  [1266] = {j1=-10.864, j2=61.673, j3=49.557, j4=-4.156, j5=76.153, j6=-10.598}
  [1267] = {j1=-10.843, j2=62.170, j3=49.109, j4=-4.208, j5=76.502, j6=-10.179}
  [1268] = {j1=-10.824, j2=62.663, j3=48.670, j4=-4.258, j5=76.846, j6=-9.764}
  [1269] = {j1=-10.807, j2=63.152, j3=48.234, j4=-4.302, j5=77.191, j6=-9.351}
  [1270] = {j1=-10.792, j2=63.641, j3=47.799, j4=-4.338, j5=77.541, j6=-8.940}
  [1271] = {j1=-10.790, j2=63.726, j3=47.722, j4=-4.344, j5=77.602, j6=-8.868}
  [1272] = {j1=-10.774, j2=64.208, j3=47.297, j4=-4.390, j5=77.944, j6=-8.456}
  [1273] = {j1=-10.750, j2=64.740, j3=46.858, j4=-4.470, j5=78.272, j6=-8.000}
  [1274] = {j1=-10.722, j2=65.202, j3=46.548, j4=-4.577, j5=78.439, j6=-7.623}
  [1275] = {j1=-10.698, j2=65.509, j3=46.425, j4=-4.679, j5=78.409, j6=-7.406}
  [1276] = {j1=-10.673, j2=65.756, j3=46.411, j4=-4.789, j5=78.237, j6=-7.269}
  [1277] = {j1=-10.648, j2=65.950, j3=46.489, j4=-4.909, j5=77.942, j6=-7.202}
  [1278] = {j1=-10.622, j2=66.101, j3=46.643, j4=-5.043, j5=77.544, j6=-7.192}
  [1279] = {j1=-10.592, j2=66.217, j3=46.855, j4=-5.194, j5=77.062, j6=-7.226}
  [1280] = {j1=-10.560, j2=66.305, j3=47.110, j4=-5.365, j5=76.516, j6=-7.293}
  [1281] = {j1=-10.559, j2=66.323, j3=47.079, j4=-5.369, j5=76.573, j6=-7.250}
  [1282] = {j1=-10.592, j2=66.234, j3=46.825, j4=-5.197, j5=77.118, j6=-7.185}
  [1283] = {j1=-10.621, j2=66.118, j3=46.614, j4=-5.046, j5=77.597, j6=-7.152}
  [1284] = {j1=-10.648, j2=65.966, j3=46.461, j4=-4.911, j5=77.993, j6=-7.164}
  [1285] = {j1=-10.673, j2=65.772, j3=46.384, j4=-4.789, j5=78.286, j6=-7.233}
  [1286] = {j1=-10.698, j2=65.525, j3=46.397, j4=-4.678, j5=78.458, j6=-7.370}
  [1287] = {j1=-10.723, j2=65.219, j3=46.519, j4=-4.575, j5=78.489, j6=-7.588}
  [1288] = {j1=-10.751, j2=64.758, j3=46.827, j4=-4.466, j5=78.325, j6=-7.964}
  [1289] = {j1=-10.775, j2=64.227, j3=47.262, j4=-4.386, j5=78.001, j6=-8.418}
  [1290] = {j1=-10.791, j2=63.747, j3=47.686, j4=-4.339, j5=77.662, j6=-8.829}
  [1291] = {j1=-10.794, j2=63.662, j3=47.761, j4=-4.333, j5=77.600, j6=-8.900}
  [1292] = {j1=-10.808, j2=63.174, j3=48.196, j4=-4.297, j5=77.252, j6=-9.311}
  [1293] = {j1=-10.825, j2=62.685, j3=48.631, j4=-4.253, j5=76.907, j6=-9.723}
  [1294] = {j1=-10.844, j2=62.192, j3=49.070, j4=-4.203, j5=76.562, j6=-10.139}
  [1295] = {j1=-10.865, j2=61.695, j3=49.519, j4=-4.150, j5=76.213, j6=-10.558}
  [1296] = {j1=-10.888, j2=61.189, j3=49.980, j4=-4.096, j5=75.855, j6=-10.983}
  [1297] = {j1=-10.912, j2=60.674, j3=50.459, j4=-4.041, j5=75.484, j6=-11.413}
  [1298] = {j1=-10.936, j2=60.147, j3=50.960, j4=-3.988, j5=75.096, j6=-11.850}
  [1299] = {j1=-10.956, j2=59.676, j3=51.416, j4=-3.950, j5=74.742, j6=-12.232}
  [1300] = {j1=-10.973, j2=59.205, j3=51.873, j4=-3.926, j5=74.393, j6=-12.600}
  [1301] = {j1=-10.987, j2=58.744, j3=52.313, j4=-3.913, j5=74.070, j6=-12.944}
  [1302] = {j1=-10.997, j2=58.303, j3=52.716, j4=-3.909, j5=73.795, j6=-13.252}
  [1303] = {j1=-10.998, j2=58.287, j3=52.730, j4=-3.909, j5=73.786, j6=-13.262}
  [1304] = {j1=-10.999, j2=58.315, j3=52.679, j4=-3.904, j5=73.859, j6=-13.219}
  [1305] = {j1=-10.998, j2=58.331, j3=52.666, j4=-3.904, j5=73.868, j6=-13.209}
  [1306] = {j1=-10.988, j2=58.771, j3=52.265, j4=-3.907, j5=74.140, j6=-12.902}
  [1307] = {j1=-10.974, j2=59.231, j3=51.828, j4=-3.920, j5=74.460, j6=-12.560}
  [1308] = {j1=-10.957, j2=59.701, j3=51.373, j4=-3.944, j5=74.807, j6=-12.193}
  [1309] = {j1=-10.937, j2=60.171, j3=50.919, j4=-3.982, j5=75.158, j6=-11.812}
  [1310] = {j1=-10.913, j2=60.697, j3=50.419, j4=-4.035, j5=75.545, j6=-11.375}
  [1311] = {j1=-10.889, j2=61.212, j3=49.940, j4=-4.090, j5=75.916, j6=-10.944}
  [1312] = {j1=-10.866, j2=61.717, j3=49.479, j4=-4.146, j5=76.274, j6=-10.519}
  [1313] = {j1=-10.845, j2=62.215, j3=49.031, j4=-4.199, j5=76.624, j6=-10.099}
  [1314] = {j1=-10.826, j2=62.707, j3=48.591, j4=-4.248, j5=76.969, j6=-9.683}
  [1315] = {j1=-10.809, j2=63.196, j3=48.158, j4=-4.292, j5=77.312, j6=-9.270}
  [1316] = {j1=-10.795, j2=63.683, j3=47.725, j4=-4.328, j5=77.659, j6=-8.861}
  [1317] = {j1=-10.793, j2=63.768, j3=47.650, j4=-4.334, j5=77.720, j6=-8.789}
  [1318] = {j1=-10.776, j2=64.246, j3=47.230, j4=-4.380, j5=78.055, j6=-8.381}
  [1319] = {j1=-10.752, j2=64.774, j3=46.798, j4=-4.462, j5=78.375, j6=-7.928}
  [1320] = {j1=-10.723, j2=65.233, j3=46.494, j4=-4.572, j5=78.535, j6=-7.553}
  [1321] = {j1=-10.699, j2=65.539, j3=46.373, j4=-4.676, j5=78.503, j6=-7.335}
  [1322] = {j1=-10.674, j2=65.785, j3=46.360, j4=-4.789, j5=78.331, j6=-7.196}
  [1323] = {j1=-10.648, j2=65.980, j3=46.438, j4=-4.912, j5=78.038, j6=-7.126}
  [1324] = {j1=-10.621, j2=66.132, j3=46.590, j4=-5.048, j5=77.643, j6=-7.113}
  [1325] = {j1=-10.591, j2=66.248, j3=46.801, j4=-5.200, j5=77.165, j6=-7.144}
  [1326] = {j1=-10.558, j2=66.337, j3=47.054, j4=-5.373, j5=76.622, j6=-7.207}
  [1327] = {j1=-10.557, j2=66.364, j3=47.008, j4=-5.379, j5=76.709, j6=-7.143}
  [1328] = {j1=-10.590, j2=66.274, j3=46.756, j4=-5.205, j5=77.248, j6=-7.082}
  [1329] = {j1=-10.620, j2=66.157, j3=46.547, j4=-5.052, j5=77.723, j6=-7.054}
  [1330] = {j1=-10.648, j2=66.004, j3=46.396, j4=-4.914, j5=78.115, j6=-7.070}
  [1331] = {j1=-10.674, j2=65.809, j3=46.319, j4=-4.789, j5=78.406, j6=-7.142}
  [1332] = {j1=-10.699, j2=65.563, j3=46.332, j4=-4.675, j5=78.577, j6=-7.282}
  [1333] = {j1=-10.724, j2=65.258, j3=46.451, j4=-4.569, j5=78.611, j6=-7.501}
  [1334] = {j1=-10.754, j2=64.801, j3=46.751, j4=-4.456, j5=78.455, j6=-7.875}
  [1335] = {j1=-10.778, j2=64.276, j3=47.178, j4=-4.373, j5=78.141, j6=-8.324}
  [1336] = {j1=-10.794, j2=63.799, j3=47.594, j4=-4.327, j5=77.809, j6=-8.731}
  [1337] = {j1=-10.797, j2=63.715, j3=47.669, j4=-4.321, j5=77.749, j6=-8.802}
  [1338] = {j1=-10.811, j2=63.229, j3=48.099, j4=-4.285, j5=77.404, j6=-9.210}
  [1339] = {j1=-10.828, j2=62.740, j3=48.533, j4=-4.241, j5=77.060, j6=-9.623}
  [1340] = {j1=-10.847, j2=62.248, j3=48.972, j4=-4.191, j5=76.714, j6=-10.039}
  [1341] = {j1=-10.868, j2=61.749, j3=49.422, j4=-4.138, j5=76.363, j6=-10.461}
  [1342] = {j1=-10.891, j2=61.244, j3=49.884, j4=-4.083, j5=76.003, j6=-10.887}
  [1343] = {j1=-10.915, j2=60.729, j3=50.363, j4=-4.027, j5=75.632, j6=-11.318}
  [1344] = {j1=-10.940, j2=60.203, j3=50.861, j4=-3.973, j5=75.246, j6=-11.755}
  [1345] = {j1=-10.960, j2=59.734, j3=51.313, j4=-3.935, j5=74.897, j6=-12.135}
  [1346] = {j1=-10.976, j2=59.266, j3=51.765, j4=-3.910, j5=74.554, j6=-12.500}
  [1347] = {j1=-10.990, j2=58.808, j3=52.199, j4=-3.898, j5=74.237, j6=-12.840}
  [1348] = {j1=-11.000, j2=58.369, j3=52.597, j4=-3.895, j5=73.967, j6=-13.144}
  [1349] = {j1=-11.000, j2=58.354, j3=52.611, j4=-3.895, j5=73.959, j6=-13.154}
  [1350] = {j1=-11.002, j2=58.398, j3=52.533, j4=-3.888, j5=74.070, j6=-13.089}
  [1351] = {j1=-11.001, j2=58.413, j3=52.520, j4=-3.888, j5=74.078, j6=-13.078}
  [1352] = {j1=-10.991, j2=58.849, j3=52.125, j4=-3.890, j5=74.344, j6=-12.777}
  [1353] = {j1=-10.978, j2=59.305, j3=51.696, j4=-3.902, j5=74.655, j6=-12.440}
  [1354] = {j1=-10.962, j2=59.771, j3=51.248, j4=-3.926, j5=74.993, j6=-12.077}
  [1355] = {j1=-10.942, j2=60.238, j3=50.800, j4=-3.964, j5=75.338, j6=-11.698}
  [1356] = {j1=-10.917, j2=60.762, j3=50.303, j4=-4.019, j5=75.722, j6=-11.262}
  [1357] = {j1=-10.893, j2=61.277, j3=49.825, j4=-4.075, j5=76.093, j6=-10.830}
  [1358] = {j1=-10.870, j2=61.783, j3=49.363, j4=-4.131, j5=76.454, j6=-10.403}
  [1359] = {j1=-10.848, j2=62.281, j3=48.913, j4=-4.184, j5=76.806, j6=-9.980}
  [1360] = {j1=-10.829, j2=62.774, j3=48.474, j4=-4.234, j5=77.152, j6=-9.562}
  [1361] = {j1=-10.812, j2=63.261, j3=48.042, j4=-4.278, j5=77.495, j6=-9.150}
  [1362] = {j1=-10.798, j2=63.746, j3=47.614, j4=-4.313, j5=77.837, j6=-8.743}
  [1363] = {j1=-10.796, j2=63.830, j3=47.539, j4=-4.319, j5=77.897, j6=-8.672}
  [1364] = {j1=-10.780, j2=64.304, j3=47.127, j4=-4.366, j5=78.224, j6=-8.268}
  [1365] = {j1=-10.755, j2=64.826, j3=46.707, j4=-4.450, j5=78.531, j6=-7.821}
  [1366] = {j1=-10.726, j2=65.281, j3=46.411, j4=-4.565, j5=78.682, j6=-7.448}
  [1367] = {j1=-10.700, j2=65.584, j3=46.295, j4=-4.673, j5=78.646, j6=-7.229}
  [1368] = {j1=-10.674, j2=65.830, j3=46.283, j4=-4.789, j5=78.474, j6=-7.088}
  [1369] = {j1=-10.648, j2=66.025, j3=46.360, j4=-4.916, j5=78.184, j6=-7.014}
  [1370] = {j1=-10.620, j2=66.178, j3=46.510, j4=-5.054, j5=77.794, j6=-6.995}
  [1371] = {j1=-10.589, j2=66.296, j3=46.718, j4=-5.210, j5=77.322, j6=-7.020}
  [1372] = {j1=-10.556, j2=66.386, j3=46.969, j4=-5.385, j5=76.785, j6=-7.078}
  [1373] = {j1=-10.555, j2=66.413, j3=46.922, j4=-5.391, j5=76.872, j6=-7.014}
  [1374] = {j1=-10.588, j2=66.322, j3=46.672, j4=-5.215, j5=77.405, j6=-6.959}
  [1375] = {j1=-10.619, j2=66.203, j3=46.466, j4=-5.058, j5=77.874, j6=-6.936}
  [1376] = {j1=-10.647, j2=66.049, j3=46.318, j4=-4.918, j5=78.261, j6=-6.957}
  [1377] = {j1=-10.674, j2=65.854, j3=46.242, j4=-4.790, j5=78.549, j6=-7.033}
  [1378] = {j1=-10.700, j2=65.608, j3=46.253, j4=-4.672, j5=78.721, j6=-7.176}
  [1379] = {j1=-10.727, j2=65.305, j3=46.368, j4=-4.561, j5=78.758, j6=-7.395}
  [1380] = {j1=-10.757, j2=64.854, j3=46.659, j4=-4.444, j5=78.612, j6=-7.766}
  [1381] = {j1=-10.782, j2=64.334, j3=47.075, j4=-4.359, j5=78.310, j6=-8.211}
  [1382] = {j1=-10.798, j2=63.862, j3=47.483, j4=-4.312, j5=77.986, j6=-8.613}
  [1383] = {j1=-10.800, j2=63.778, j3=47.557, j4=-4.306, j5=77.927, j6=-8.683}
  [1384] = {j1=-10.814, j2=63.294, j3=47.984, j4=-4.271, j5=77.586, j6=-9.090}
  [1385] = {j1=-10.831, j2=62.806, j3=48.416, j4=-4.227, j5=77.243, j6=-9.502}
  [1386] = {j1=-10.850, j2=62.313, j3=48.856, j4=-4.177, j5=76.895, j6=-9.921}
  [1387] = {j1=-10.871, j2=61.814, j3=49.307, j4=-4.123, j5=76.540, j6=-10.345}
  [1388] = {j1=-10.894, j2=61.308, j3=49.770, j4=-4.067, j5=76.178, j6=-10.773}
  [1389] = {j1=-10.919, j2=60.793, j3=50.249, j4=-4.010, j5=75.807, j6=-11.206}
  [1390] = {j1=-10.944, j2=60.269, j3=50.744, j4=-3.955, j5=75.424, j6=-11.642}
  [1391] = {j1=-10.964, j2=59.804, j3=51.189, j4=-3.916, j5=75.082, j6=-12.019}
  [1392] = {j1=-10.981, j2=59.340, j3=51.633, j4=-3.892, j5=74.748, j6=-12.379}
  [1393] = {j1=-10.993, j2=58.886, j3=52.059, j4=-3.880, j5=74.441, j6=-12.713}
  [1394] = {j1=-11.003, j2=58.452, j3=52.449, j4=-3.880, j5=74.180, j6=-13.011}
  [1395] = {j1=-11.003, j2=58.437, j3=52.463, j4=-3.880, j5=74.171, j6=-13.022}
  [1396] = {j1=-11.004, j2=58.482, j3=52.382, j4=-3.872, j5=74.286, j6=-12.953}
  [1397] = {j1=-11.004, j2=58.497, j3=52.369, j4=-3.872, j5=74.294, j6=-12.943}
  [1398] = {j1=-10.995, j2=58.929, j3=51.983, j4=-3.872, j5=74.550, j6=-12.648}
  [1399] = {j1=-10.982, j2=59.380, j3=51.563, j4=-3.883, j5=74.851, j6=-12.317}
  [1400] = {j1=-10.966, j2=59.841, j3=51.124, j4=-3.907, j5=75.179, j6=-11.961}
  [1401] = {j1=-10.946, j2=60.303, j3=50.683, j4=-3.947, j5=75.516, j6=-11.585}
  [1402] = {j1=-10.921, j2=60.826, j3=50.190, j4=-4.002, j5=75.896, j6=-11.150}
  [1403] = {j1=-10.896, j2=61.340, j3=49.713, j4=-4.059, j5=76.267, j6=-10.717}
  [1404] = {j1=-10.873, j2=61.847, j3=49.250, j4=-4.116, j5=76.629, j6=-10.287}
  [1405] = {j1=-10.852, j2=62.346, j3=48.798, j4=-4.170, j5=76.985, j6=-9.862}
  [1406] = {j1=-10.833, j2=62.839, j3=48.358, j4=-4.220, j5=77.334, j6=-9.442}
  [1407] = {j1=-10.816, j2=63.327, j3=47.926, j4=-4.263, j5=77.677, j6=-9.029}
  [1408] = {j1=-10.802, j2=63.809, j3=47.502, j4=-4.299, j5=78.015, j6=-8.624}
  [1409] = {j1=-10.800, j2=63.893, j3=47.429, j4=-4.305, j5=78.074, j6=-8.554}
  [1410] = {j1=-10.784, j2=64.362, j3=47.025, j4=-4.352, j5=78.392, j6=-8.154}
  [1411] = {j1=-10.759, j2=64.879, j3=46.615, j4=-4.438, j5=78.687, j6=-7.712}
  [1412] = {j1=-10.728, j2=65.328, j3=46.329, j4=-4.557, j5=78.828, j6=-7.342}
  [1413] = {j1=-10.701, j2=65.629, j3=46.216, j4=-4.670, j5=78.789, j6=-7.122}
  [1414] = {j1=-10.674, j2=65.874, j3=46.206, j4=-4.790, j5=78.617, j6=-6.978}
  [1415] = {j1=-10.647, j2=66.070, j3=46.282, j4=-4.919, j5=78.330, j6=-6.900}
  [1416] = {j1=-10.619, j2=66.224, j3=46.430, j4=-5.061, j5=77.944, j6=-6.876}
  [1417] = {j1=-10.588, j2=66.344, j3=46.635, j4=-5.219, j5=77.478, j6=-6.896}
  [1418] = {j1=-10.554, j2=66.436, j3=46.883, j4=-5.396, j5=76.948, j6=-6.949}
  [1419] = {j1=-10.552, j2=66.463, j3=46.836, j4=-5.403, j5=77.036, j6=-6.883}
  [1420] = {j1=-10.587, j2=66.370, j3=46.589, j4=-5.224, j5=77.563, j6=-6.834}
  [1421] = {j1=-10.618, j2=66.250, j3=46.386, j4=-5.065, j5=78.025, j6=-6.817}
  [1422] = {j1=-10.647, j2=66.095, j3=46.240, j4=-4.921, j5=78.407, j6=-6.843}
  [1423] = {j1=-10.675, j2=65.898, j3=46.164, j4=-4.790, j5=78.692, j6=-6.924}
  [1424] = {j1=-10.702, j2=65.653, j3=46.174, j4=-4.668, j5=78.863, j6=-7.069}
  [1425] = {j1=-10.729, j2=65.353, j3=46.285, j4=-4.554, j5=78.904, j6=-7.289}
  [1426] = {j1=-10.760, j2=64.906, j3=46.568, j4=-4.433, j5=78.768, j6=-7.657}
  [1427] = {j1=-10.785, j2=64.392, j3=46.973, j4=-4.345, j5=78.478, j6=-8.096}
  [1428] = {j1=-10.802, j2=63.925, j3=47.373, j4=-4.297, j5=78.163, j6=-8.494}
  [1429] = {j1=-10.804, j2=63.841, j3=47.446, j4=-4.292, j5=78.105, j6=-8.564}
  [1430] = {j1=-10.818, j2=63.359, j3=47.869, j4=-4.256, j5=77.767, j6=-8.969}
  [1431] = {j1=-10.834, j2=62.872, j3=48.301, j4=-4.213, j5=77.423, j6=-9.382}
  [1432] = {j1=-10.854, j2=62.378, j3=48.743, j4=-4.163, j5=77.072, j6=-9.803}
  [1433] = {j1=-10.875, j2=61.877, j3=49.196, j4=-4.108, j5=76.714, j6=-10.230}
  [1434] = {j1=-10.898, j2=61.370, j3=49.660, j4=-4.051, j5=76.349, j6=-10.661}
  [1435] = {j1=-10.923, j2=60.856, j3=50.138, j4=-3.994, j5=75.978, j6=-11.095}
  [1436] = {j1=-10.948, j2=60.334, j3=50.628, j4=-3.937, j5=75.600, j6=-11.529}
  [1437] = {j1=-10.968, j2=59.873, j3=51.066, j4=-3.898, j5=75.266, j6=-11.902}
  [1438] = {j1=-10.985, j2=59.415, j3=51.500, j4=-3.874, j5=74.944, j6=-12.255}
  [1439] = {j1=-10.997, j2=58.967, j3=51.915, j4=-3.863, j5=74.649, j6=-12.582}
  [1440] = {j1=-11.006, j2=58.537, j3=52.297, j4=-3.864, j5=74.397, j6=-12.874}
  [1441] = {j1=-11.006, j2=58.522, j3=52.311, j4=-3.864, j5=74.388, j6=-12.884}
  [1442] = {j1=-11.007, j2=58.569, j3=52.226, j4=-3.857, j5=74.507, j6=-12.814}
  [1443] = {j1=-11.007, j2=58.584, j3=52.214, j4=-3.857, j5=74.514, j6=-12.804}
  [1444] = {j1=-10.998, j2=59.011, j3=51.837, j4=-3.855, j5=74.760, j6=-12.516}
  [1445] = {j1=-10.986, j2=59.455, j3=51.428, j4=-3.865, j5=75.048, j6=-12.193}
  [1446] = {j1=-10.970, j2=59.910, j3=51.001, j4=-3.889, j5=75.363, j6=-11.843}
  [1447] = {j1=-10.950, j2=60.368, j3=50.568, j4=-3.929, j5=75.691, j6=-11.473}
  [1448] = {j1=-10.925, j2=60.888, j3=50.081, j4=-3.986, j5=76.065, j6=-11.040}
  [1449] = {j1=-10.900, j2=61.402, j3=49.605, j4=-4.044, j5=76.435, j6=-10.606}
  [1450] = {j1=-10.877, j2=61.909, j3=49.140, j4=-4.101, j5=76.801, j6=-10.173}
  [1451] = {j1=-10.855, j2=62.410, j3=48.686, j4=-4.155, j5=77.160, j6=-9.745}
  [1452] = {j1=-10.836, j2=62.904, j3=48.244, j4=-4.205, j5=77.512, j6=-9.322}
  [1453] = {j1=-10.819, j2=63.392, j3=47.812, j4=-4.249, j5=77.857, j6=-8.908}
  [1454] = {j1=-10.806, j2=63.872, j3=47.391, j4=-4.284, j5=78.192, j6=-8.504}
  [1455] = {j1=-10.803, j2=63.955, j3=47.320, j4=-4.290, j5=78.249, j6=-8.434}
  [1456] = {j1=-10.787, j2=64.420, j3=46.923, j4=-4.338, j5=78.559, j6=-8.039}
  [1457] = {j1=-10.762, j2=64.931, j3=46.524, j4=-4.427, j5=78.843, j6=-7.602}
  [1458] = {j1=-10.730, j2=65.375, j3=46.247, j4=-4.550, j5=78.974, j6=-7.235}
  [1459] = {j1=-10.702, j2=65.674, j3=46.138, j4=-4.666, j5=78.930, j6=-7.015}
  [1460] = {j1=-10.675, j2=65.918, j3=46.129, j4=-4.790, j5=78.759, j6=-6.868}
  [1461] = {j1=-10.647, j2=66.115, j3=46.205, j4=-4.922, j5=78.475, j6=-6.786}
  [1462] = {j1=-10.618, j2=66.270, j3=46.350, j4=-5.067, j5=78.095, j6=-6.757}
  [1463] = {j1=-10.586, j2=66.392, j3=46.552, j4=-5.227, j5=77.635, j6=-6.771}
  [1464] = {j1=-10.552, j2=66.485, j3=46.798, j4=-5.407, j5=77.110, j6=-6.818}
  [1465] = {j1=-10.550, j2=66.513, j3=46.749, j4=-5.413, j5=77.199, j6=-6.752}
  [1466] = {j1=-10.585, j2=66.419, j3=46.506, j4=-5.232, j5=77.720, j6=-6.708}
  [1467] = {j1=-10.617, j2=66.296, j3=46.306, j4=-5.071, j5=78.176, j6=-6.697}
  [1468] = {j1=-10.647, j2=66.140, j3=46.162, j4=-4.924, j5=78.553, j6=-6.728}
  [1469] = {j1=-10.675, j2=65.943, j3=46.087, j4=-4.790, j5=78.834, j6=-6.813}
  [1470] = {j1=-10.703, j2=65.698, j3=46.096, j4=-4.665, j5=79.005, j6=-6.961}
  [1471] = {j1=-10.731, j2=65.400, j3=46.203, j4=-4.546, j5=79.050, j6=-7.181}
  [1472] = {j1=-10.763, j2=64.958, j3=46.476, j4=-4.421, j5=78.923, j6=-7.547}
  [1473] = {j1=-10.789, j2=64.450, j3=46.871, j4=-4.331, j5=78.645, j6=-7.981}
  [1474] = {j1=-10.805, j2=63.987, j3=47.264, j4=-4.283, j5=78.338, j6=-8.374}
  [1475] = {j1=-10.807, j2=63.904, j3=47.336, j4=-4.277, j5=78.281, j6=-8.444}
  [1476] = {j1=-10.821, j2=63.423, j3=47.756, j4=-4.242, j5=77.946, j6=-8.847}
  [1477] = {j1=-10.838, j2=62.935, j3=48.188, j4=-4.198, j5=77.600, j6=-9.263}
  [1478] = {j1=-10.857, j2=62.440, j3=48.632, j4=-4.148, j5=77.245, j6=-9.687}
  [1479] = {j1=-10.879, j2=61.938, j3=49.088, j4=-4.093, j5=76.882, j6=-10.117}
  [1480] = {j1=-10.902, j2=61.430, j3=49.554, j4=-4.035, j5=76.515, j6=-10.551}
  [1481] = {j1=-10.927, j2=60.916, j3=50.030, j4=-3.977, j5=76.144, j6=-10.985}
  [1482] = {j1=-10.952, j2=60.398, j3=50.515, j4=-3.920, j5=75.772, j6=-11.417}
  [1483] = {j1=-10.972, j2=59.942, j3=50.944, j4=-3.880, j5=75.450, j6=-11.784}
  [1484] = {j1=-10.988, j2=59.490, j3=51.366, j4=-3.856, j5=75.141, j6=-12.130}
  [1485] = {j1=-11.000, j2=59.049, j3=51.769, j4=-3.846, j5=74.859, j6=-12.448}
  [1486] = {j1=-11.008, j2=58.625, j3=52.141, j4=-3.848, j5=74.619, j6=-12.733}
  [1487] = {j1=-11.009, j2=58.610, j3=52.154, j4=-3.848, j5=74.610, j6=-12.743}
  [1488] = {j1=-11.010, j2=58.659, j3=52.067, j4=-3.841, j5=74.732, j6=-12.670}
  [1489] = {j1=-11.009, j2=58.674, j3=52.054, j4=-3.841, j5=74.739, j6=-12.660}
  [1490] = {j1=-11.002, j2=59.094, j3=51.689, j4=-3.838, j5=74.973, j6=-12.380}
  [1491] = {j1=-10.990, j2=59.531, j3=51.293, j4=-3.847, j5=75.246, j6=-12.066}
  [1492] = {j1=-10.974, j2=59.979, j3=50.878, j4=-3.871, j5=75.546, j6=-11.724}
  [1493] = {j1=-10.954, j2=60.432, j3=50.455, j4=-3.911, j5=75.862, j6=-11.360}
  [1494] = {j1=-10.929, j2=60.948, j3=49.974, j4=-3.969, j5=76.230, j6=-10.930}
  [1495] = {j1=-10.904, j2=61.461, j3=49.500, j4=-4.027, j5=76.599, j6=-10.496}
  [1496] = {j1=-10.881, j2=61.969, j3=49.033, j4=-4.085, j5=76.968, j6=-10.061}
  [1497] = {j1=-10.859, j2=62.472, j3=48.577, j4=-4.140, j5=77.331, j6=-9.629}
  [1498] = {j1=-10.839, j2=62.967, j3=48.132, j4=-4.191, j5=77.688, j6=-9.203}
  [1499] = {j1=-10.823, j2=63.455, j3=47.700, j4=-4.234, j5=78.034, j6=-8.787}
  [1500] = {j1=-10.809, j2=63.935, j3=47.282, j4=-4.270, j5=78.367, j6=-8.383}
  [1501] = {j1=-10.807, j2=64.017, j3=47.211, j4=-4.275, j5=78.424, j6=-8.314}
  [1502] = {j1=-10.791, j2=64.478, j3=46.822, j4=-4.324, j5=78.725, j6=-7.923}
  [1503] = {j1=-10.765, j2=64.982, j3=46.434, j4=-4.415, j5=78.997, j6=-7.491}
  [1504] = {j1=-10.732, j2=65.422, j3=46.166, j4=-4.542, j5=79.118, j6=-7.127}
  [1505] = {j1=-10.704, j2=65.719, j3=46.061, j4=-4.663, j5=79.072, j6=-6.906}
  [1506] = {j1=-10.675, j2=65.962, j3=46.053, j4=-4.789, j5=78.900, j6=-6.757}
  [1507] = {j1=-10.647, j2=66.159, j3=46.127, j4=-4.925, j5=78.619, j6=-6.671}
  [1508] = {j1=-10.617, j2=66.316, j3=46.271, j4=-5.073, j5=78.244, j6=-6.637}
  [1509] = {j1=-10.585, j2=66.440, j3=46.470, j4=-5.236, j5=77.791, j6=-6.645}
  [1510] = {j1=-10.550, j2=66.535, j3=46.712, j4=-5.418, j5=77.273, j6=-6.686}
  [1511] = {j1=-10.548, j2=66.563, j3=46.663, j4=-5.424, j5=77.363, j6=-6.620}
  [1512] = {j1=-10.584, j2=66.467, j3=46.422, j4=-5.241, j5=77.877, j6=-6.582}
  [1513] = {j1=-10.616, j2=66.342, j3=46.225, j4=-5.076, j5=78.326, j6=-6.576}
  [1514] = {j1=-10.646, j2=66.184, j3=46.084, j4=-4.927, j5=78.698, j6=-6.613}
  [1515] = {j1=-10.675, j2=65.987, j3=46.011, j4=-4.790, j5=78.976, j6=-6.701}
  [1516] = {j1=-10.704, j2=65.743, j3=46.019, j4=-4.661, j5=79.147, j6=-6.852}
  [1517] = {j1=-10.733, j2=65.447, j3=46.122, j4=-4.539, j5=79.194, j6=-7.073}
  [1518] = {j1=-10.766, j2=65.010, j3=46.386, j4=-4.410, j5=79.077, j6=-7.435}
  [1519] = {j1=-10.792, j2=64.508, j3=46.770, j4=-4.317, j5=78.810, j6=-7.864}
  [1520] = {j1=-10.809, j2=64.048, j3=47.156, j4=-4.268, j5=78.511, j6=-8.254}
  [1521] = {j1=-10.811, j2=63.966, j3=47.227, j4=-4.263, j5=78.455, j6=-8.323}
  [1522] = {j1=-10.824, j2=63.487, j3=47.645, j4=-4.227, j5=78.122, j6=-8.727}
  [1523] = {j1=-10.841, j2=62.998, j3=48.078, j4=-4.183, j5=77.773, j6=-9.144}
  [1524] = {j1=-10.861, j2=62.501, j3=48.525, j4=-4.132, j5=77.414, j6=-9.572}
  [1525] = {j1=-10.883, j2=61.997, j3=48.984, j4=-4.077, j5=77.047, j6=-10.005}
  [1526] = {j1=-10.906, j2=61.488, j3=49.452, j4=-4.019, j5=76.676, j6=-10.442}
  [1527] = {j1=-10.931, j2=60.975, j3=49.926, j4=-3.960, j5=76.306, j6=-10.876}
  [1528] = {j1=-10.956, j2=60.460, j3=50.404, j4=-3.902, j5=75.942, j6=-11.304}
  [1529] = {j1=-10.977, j2=60.011, j3=50.822, j4=-3.862, j5=75.632, j6=-11.664}
  [1530] = {j1=-10.992, j2=59.566, j3=51.230, j4=-3.838, j5=75.339, j6=-12.001}
  [1531] = {j1=-11.004, j2=59.133, j3=51.620, j4=-3.829, j5=75.073, j6=-12.310}
  [1532] = {j1=-11.011, j2=58.715, j3=51.980, j4=-3.832, j5=74.845, j6=-12.587}
  [1533] = {j1=-11.011, j2=58.700, j3=51.993, j4=-3.833, j5=74.837, j6=-12.597}
  [1534] = {j1=-11.012, j2=58.746, j3=51.911, j4=-3.827, j5=74.952, j6=-12.528}
  [1535] = {j1=-11.012, j2=58.761, j3=51.899, j4=-3.826, j5=74.958, j6=-12.519}
  [1536] = {j1=-11.005, j2=59.175, j3=51.545, j4=-3.822, j5=75.179, j6=-12.246}
  [1537] = {j1=-10.994, j2=59.604, j3=51.163, j4=-3.831, j5=75.436, j6=-11.942}
  [1538] = {j1=-10.978, j2=60.044, j3=50.762, j4=-3.854, j5=75.720, j6=-11.610}
  [1539] = {j1=-10.958, j2=60.491, j3=50.351, j4=-3.895, j5=76.023, j6=-11.253}
  [1540] = {j1=-10.933, j2=61.003, j3=49.877, j4=-3.953, j5=76.382, j6=-10.827}
  [1541] = {j1=-10.908, j2=61.515, j3=49.404, j4=-4.012, j5=76.751, j6=-10.392}
  [1542] = {j1=-10.884, j2=62.024, j3=48.936, j4=-4.070, j5=77.121, j6=-9.955}
  [1543] = {j1=-10.863, j2=62.528, j3=48.477, j4=-4.126, j5=77.490, j6=-9.520}
  [1544] = {j1=-10.843, j2=63.026, j3=48.029, j4=-4.176, j5=77.851, j6=-9.090}
  [1545] = {j1=-10.826, j2=63.514, j3=47.596, j4=-4.220, j5=78.200, j6=-8.672}
  [1546] = {j1=-10.812, j2=63.993, j3=47.180, j4=-4.256, j5=78.532, j6=-8.268}
  [1547] = {j1=-10.810, j2=64.075, j3=47.110, j4=-4.261, j5=78.587, j6=-8.200}
  [1548] = {j1=-10.794, j2=64.532, j3=46.727, j4=-4.311, j5=78.882, j6=-7.811}
  [1549] = {j1=-10.768, j2=65.031, j3=46.349, j4=-4.404, j5=79.142, j6=-7.384}
  [1550] = {j1=-10.734, j2=65.466, j3=46.089, j4=-4.535, j5=79.255, j6=-7.023}
  [1551] = {j1=-10.705, j2=65.761, j3=45.988, j4=-4.659, j5=79.205, j6=-6.801}
  [1552] = {j1=-10.676, j2=66.004, j3=45.981, j4=-4.789, j5=79.034, j6=-6.650}
  [1553] = {j1=-10.647, j2=66.202, j3=46.054, j4=-4.928, j5=78.756, j6=-6.560}
  [1554] = {j1=-10.616, j2=66.360, j3=46.195, j4=-5.078, j5=78.386, j6=-6.521}
  [1555] = {j1=-10.583, j2=66.485, j3=46.391, j4=-5.243, j5=77.939, j6=-6.524}
  [1556] = {j1=-10.548, j2=66.582, j3=46.631, j4=-5.428, j5=77.427, j6=-6.559}
  [1557] = {j1=-10.547, j2=66.608, j3=46.585, j4=-5.433, j5=77.510, j6=-6.498}
  [1558] = {j1=-10.583, j2=66.510, j3=46.348, j4=-5.247, j5=78.017, j6=-6.465}
  [1559] = {j1=-10.615, j2=66.384, j3=46.154, j4=-5.081, j5=78.461, j6=-6.465}
  [1560] = {j1=-10.646, j2=66.224, j3=46.015, j4=-4.929, j5=78.828, j6=-6.506}
  [1561] = {j1=-10.676, j2=66.026, j3=45.942, j4=-4.789, j5=79.103, j6=-6.599}
  [1562] = {j1=-10.705, j2=65.783, j3=45.950, j4=-4.658, j5=79.273, j6=-6.751}
  [1563] = {j1=-10.735, j2=65.488, j3=46.050, j4=-4.532, j5=79.323, j6=-6.973}
  [1564] = {j1=-10.769, j2=65.055, j3=46.306, j4=-4.399, j5=79.214, j6=-7.333}
  [1565] = {j1=-10.796, j2=64.558, j3=46.681, j4=-4.304, j5=78.958, j6=-7.758}
  [1566] = {j1=-10.812, j2=64.102, j3=47.061, j4=-4.255, j5=78.665, j6=-8.145}
  [1567] = {j1=-10.814, j2=64.020, j3=47.132, j4=-4.249, j5=78.609, j6=-8.214}
  [1568] = {j1=-10.828, j2=63.542, j3=47.547, j4=-4.213, j5=78.277, j6=-8.617}
  [1569] = {j1=-10.845, j2=63.052, j3=47.982, j4=-4.169, j5=77.926, j6=-9.037}
  [1570] = {j1=-10.864, j2=62.554, j3=48.432, j4=-4.118, j5=77.561, j6=-9.468}
  [1571] = {j1=-10.886, j2=62.048, j3=48.894, j4=-4.062, j5=77.190, j6=-9.905}
  [1572] = {j1=-10.910, j2=61.538, j3=49.363, j4=-4.004, j5=76.817, j6=-10.344}
  [1573] = {j1=-10.935, j2=61.026, j3=49.836, j4=-3.944, j5=76.449, j6=-10.778}
  [1574] = {j1=-10.960, j2=60.515, j3=50.307, j4=-3.886, j5=76.092, j6=-11.202}
  [1575] = {j1=-10.980, j2=60.072, j3=50.713, j4=-3.846, j5=75.795, j6=-11.555}
  [1576] = {j1=-10.996, j2=59.635, j3=51.108, j4=-3.822, j5=75.518, j6=-11.882}
  [1577] = {j1=-11.006, j2=59.210, j3=51.483, j4=-3.813, j5=75.269, j6=-12.181}
  [1578] = {j1=-11.013, j2=58.799, j3=51.832, j4=-3.818, j5=75.054, j6=-12.450}
  [1579] = {j1=-11.013, j2=58.784, j3=51.844, j4=-3.818, j5=75.047, j6=-12.459}
  [1580] = {j1=-11.014, j2=58.831, j3=51.759, j4=-3.812, j5=75.164, j6=-12.389}
  [1581] = {j1=-11.014, j2=58.846, j3=51.748, j4=-3.812, j5=75.170, j6=-12.380}
  [1582] = {j1=-11.007, j2=59.253, j3=51.406, j4=-3.807, j5=75.377, j6=-12.116}
  [1583] = {j1=-10.997, j2=59.674, j3=51.039, j4=-3.815, j5=75.616, j6=-11.822}
  [1584] = {j1=-10.982, j2=60.106, j3=50.653, j4=-3.838, j5=75.883, j6=-11.499}
  [1585] = {j1=-10.962, j2=60.545, j3=50.254, j4=-3.879, j5=76.172, j6=-11.150}
  [1586] = {j1=-10.937, j2=61.053, j3=49.788, j4=-3.937, j5=76.523, j6=-10.729}
  [1587] = {j1=-10.912, j2=61.564, j3=49.318, j4=-3.996, j5=76.889, j6=-10.295}
  [1588] = {j1=-10.888, j2=62.074, j3=48.848, j4=-4.055, j5=77.262, j6=-9.856}
  [1589] = {j1=-10.866, j2=62.580, j3=48.386, j4=-4.111, j5=77.635, j6=-9.417}
  [1590] = {j1=-10.846, j2=63.079, j3=47.935, j4=-4.162, j5=78.001, j6=-8.984}
  [1591] = {j1=-10.829, j2=63.569, j3=47.500, j4=-4.206, j5=78.353, j6=-8.563}
  [1592] = {j1=-10.816, j2=64.046, j3=47.085, j4=-4.242, j5=78.685, j6=-8.159}
  [1593] = {j1=-10.814, j2=64.128, j3=47.016, j4=-4.248, j5=78.739, j6=-8.090}
  [1594] = {j1=-10.797, j2=64.582, j3=46.639, j4=-4.298, j5=79.028, j6=-7.705}
  [1595] = {j1=-10.770, j2=65.076, j3=46.270, j4=-4.393, j5=79.279, j6=-7.282}
  [1596] = {j1=-10.736, j2=65.507, j3=46.018, j4=-4.528, j5=79.382, j6=-6.923}
  [1597] = {j1=-10.706, j2=65.800, j3=45.920, j4=-4.655, j5=79.330, j6=-6.701}
  [1598] = {j1=-10.676, j2=66.043, j3=45.914, j4=-4.788, j5=79.159, j6=-6.547}
  [1599] = {j1=-10.646, j2=66.241, j3=45.986, j4=-4.930, j5=78.885, j6=-6.453}
  [1600] = {j1=-10.615, j2=66.401, j3=46.125, j4=-5.082, j5=78.520, j6=-6.409}
  [1601] = {j1=-10.582, j2=66.527, j3=46.318, j4=-5.250, j5=78.078, j6=-6.407}
  [1602] = {j1=-10.546, j2=66.626, j3=46.554, j4=-5.436, j5=77.574, j6=-6.437}
  [1603] = {j1=-10.545, j2=66.652, j3=46.508, j4=-5.441, j5=77.657, j6=-6.375}
  [1604] = {j1=-10.581, j2=66.553, j3=46.274, j4=-5.254, j5=78.158, j6=-6.348}
  [1605] = {j1=-10.615, j2=66.425, j3=46.083, j4=-5.085, j5=78.595, j6=-6.353}
  [1606] = {j1=-10.646, j2=66.264, j3=45.946, j4=-4.931, j5=78.957, j6=-6.399}
  [1607] = {j1=-10.676, j2=66.065, j3=45.875, j4=-4.788, j5=79.229, j6=-6.495}
  [1608] = {j1=-10.707, j2=65.822, j3=45.882, j4=-4.654, j5=79.398, j6=-6.650}
  [1609] = {j1=-10.737, j2=65.529, j3=45.979, j4=-4.525, j5=79.451, j6=-6.872}
  [1610] = {j1=-10.772, j2=65.100, j3=46.228, j4=-4.389, j5=79.350, j6=-7.230}
  [1611] = {j1=-10.799, j2=64.608, j3=46.594, j4=-4.292, j5=79.103, j6=-7.651}
  [1612] = {j1=-10.815, j2=64.155, j3=46.968, j4=-4.241, j5=78.816, j6=-8.036}
  [1613] = {j1=-10.817, j2=64.073, j3=47.038, j4=-4.235, j5=78.761, j6=-8.104}
  [1614] = {j1=-10.831, j2=63.596, j3=47.453, j4=-4.199, j5=78.429, j6=-8.508}
  [1615] = {j1=-10.848, j2=63.105, j3=47.890, j4=-4.155, j5=78.074, j6=-8.931}
  [1616] = {j1=-10.868, j2=62.604, j3=48.344, j4=-4.103, j5=77.704, j6=-9.366}
  [1617] = {j1=-10.890, j2=62.097, j3=48.809, j4=-4.047, j5=77.328, j6=-9.807}
  [1618] = {j1=-10.914, j2=61.586, j3=49.279, j4=-3.988, j5=76.952, j6=-10.247}
  [1619] = {j1=-10.939, j2=61.075, j3=49.749, j4=-3.929, j5=76.586, j6=-10.680}
  [1620] = {j1=-10.964, j2=60.569, j3=50.212, j4=-3.870, j5=76.239, j6=-11.099}
  [1621] = {j1=-10.984, j2=60.133, j3=50.605, j4=-3.830, j5=75.957, j6=-11.444}
  [1622] = {j1=-10.999, j2=59.705, j3=50.984, j4=-3.806, j5=75.698, j6=-11.761}
  [1623] = {j1=-11.009, j2=59.288, j3=51.344, j4=-3.798, j5=75.467, j6=-12.049}
  [1624] = {j1=-11.015, j2=58.884, j3=51.680, j4=-3.804, j5=75.267, j6=-12.309}
  [1625] = {j1=-11.016, j2=58.869, j3=51.692, j4=-3.804, j5=75.259, j6=-12.318}
  [1626] = {j1=-11.016, j2=58.918, j3=51.605, j4=-3.799, j5=75.379, j6=-12.246}
  [1627] = {j1=-11.016, j2=58.932, j3=51.594, j4=-3.798, j5=75.385, j6=-12.237}
  [1628] = {j1=-11.010, j2=59.332, j3=51.265, j4=-3.792, j5=75.577, j6=-11.982}
  [1629] = {j1=-11.000, j2=59.744, j3=50.915, j4=-3.799, j5=75.797, j6=-11.699}
  [1630] = {j1=-10.985, j2=60.166, j3=50.546, j4=-3.823, j5=76.045, j6=-11.388}
  [1631] = {j1=-10.966, j2=60.599, j3=50.160, j4=-3.863, j5=76.318, j6=-11.048}
  [1632] = {j1=-10.941, j2=61.102, j3=49.702, j4=-3.921, j5=76.659, j6=-10.632}
  [1633] = {j1=-10.916, j2=61.611, j3=49.235, j4=-3.981, j5=77.022, j6=-10.199}
  [1634] = {j1=-10.892, j2=62.121, j3=48.765, j4=-4.040, j5=77.398, j6=-9.758}
  [1635] = {j1=-10.870, j2=62.629, j3=48.299, j4=-4.096, j5=77.776, j6=-9.315}
  [1636] = {j1=-10.850, j2=63.131, j3=47.844, j4=-4.147, j5=78.147, j6=-8.878}
  [1637] = {j1=-10.833, j2=63.622, j3=47.407, j4=-4.192, j5=78.503, j6=-8.454}
  [1638] = {j1=-10.819, j2=64.099, j3=46.993, j4=-4.228, j5=78.834, j6=-8.050}
  [1639] = {j1=-10.817, j2=64.180, j3=46.925, j4=-4.234, j5=78.888, j6=-7.982}
  [1640] = {j1=-10.801, j2=64.631, j3=46.554, j4=-4.285, j5=79.171, j6=-7.598}
  [1641] = {j1=-10.773, j2=65.121, j3=46.192, j4=-4.383, j5=79.413, j6=-7.179}
  [1642] = {j1=-10.738, j2=65.547, j3=45.948, j4=-4.521, j5=79.509, j6=-6.822}
  [1643] = {j1=-10.707, j2=65.839, j3=45.853, j4=-4.651, j5=79.454, j6=-6.600}
  [1644] = {j1=-10.677, j2=66.081, j3=45.847, j4=-4.787, j5=79.284, j6=-6.443}
  [1645] = {j1=-10.646, j2=66.280, j3=45.918, j4=-4.931, j5=79.013, j6=-6.345}
  [1646] = {j1=-10.615, j2=66.441, j3=46.054, j4=-5.086, j5=78.653, j6=-6.297}
  [1647] = {j1=-10.581, j2=66.570, j3=46.244, j4=-5.256, j5=78.217, j6=-6.289}
  [1648] = {j1=-10.545, j2=66.670, j3=46.477, j4=-5.444, j5=77.719, j6=-6.313}
  [1649] = {j1=-10.543, j2=66.708, j3=46.412, j4=-5.452, j5=77.837, j6=-6.227}
  [1650] = {j1=-10.580, j2=66.606, j3=46.182, j4=-5.262, j5=78.330, j6=-6.206}
  [1651] = {j1=-10.614, j2=66.476, j3=45.994, j4=-5.090, j5=78.760, j6=-6.218}
  [1652] = {j1=-10.646, j2=66.313, j3=45.861, j4=-4.933, j5=79.115, j6=-6.270}
  [1653] = {j1=-10.677, j2=66.113, j3=45.791, j4=-4.787, j5=79.383, j6=-6.370}
  [1654] = {j1=-10.708, j2=65.871, j3=45.797, j4=-4.649, j5=79.552, j6=-6.528}
  [1655] = {j1=-10.739, j2=65.580, j3=45.891, j4=-4.517, j5=79.607, j6=-6.751}
  [1656] = {j1=-10.775, j2=65.155, j3=46.131, j4=-4.376, j5=79.515, j6=-7.107}
  [1657] = {j1=-10.803, j2=64.669, j3=46.488, j4=-4.277, j5=79.278, j6=-7.524}
  [1658] = {j1=-10.819, j2=64.219, j3=46.856, j4=-4.225, j5=78.998, j6=-7.906}
  [1659] = {j1=-10.821, j2=64.137, j3=46.926, j4=-4.219, j5=78.943, j6=-7.974}
  [1660] = {j1=-10.835, j2=63.660, j3=47.340, j4=-4.183, j5=78.610, j6=-8.379}
  [1661] = {j1=-10.852, j2=63.167, j3=47.780, j4=-4.137, j5=78.250, j6=-8.806}
  [1662] = {j1=-10.873, j2=62.664, j3=48.238, j4=-4.085, j5=77.874, j6=-9.246}
  [1663] = {j1=-10.895, j2=62.154, j3=48.707, j4=-4.029, j5=77.491, j6=-9.691}
  [1664] = {j1=-10.919, j2=61.643, j3=49.179, j4=-3.970, j5=77.113, j6=-10.133}
  [1665] = {j1=-10.943, j2=61.134, j3=49.645, j4=-3.910, j5=76.751, j6=-10.565}
  [1666] = {j1=-10.969, j2=60.634, j3=50.097, j4=-3.852, j5=76.417, j6=-10.977}
  [1667] = {j1=-10.988, j2=60.207, j3=50.473, j4=-3.811, j5=76.154, j6=-11.310}
  [1668] = {j1=-11.002, j2=59.791, j3=50.831, j4=-3.788, j5=75.920, j6=-11.613}
  [1669] = {j1=-11.012, j2=59.385, j3=51.170, j4=-3.781, j5=75.713, j6=-11.887}
  [1670] = {j1=-11.018, j2=58.991, j3=51.489, j4=-3.788, j5=75.531, j6=-12.136}
  [1671] = {j1=-11.018, j2=58.976, j3=51.501, j4=-3.788, j5=75.524, j6=-12.144}
  [1672] = {j1=-11.018, j2=59.011, j3=51.440, j4=-3.784, j5=75.608, j6=-12.094}
  [1673] = {j1=-11.018, j2=59.024, j3=51.430, j4=-3.784, j5=75.613, j6=-12.085}
  [1674] = {j1=-11.013, j2=59.416, j3=51.116, j4=-3.777, j5=75.788, j6=-11.840}
  [1675] = {j1=-11.003, j2=59.817, j3=50.784, j4=-3.784, j5=75.987, j6=-11.570}
  [1676] = {j1=-10.989, j2=60.230, j3=50.433, j4=-3.807, j5=76.213, j6=-11.271}
  [1677] = {j1=-10.970, j2=60.653, j3=50.063, j4=-3.847, j5=76.469, j6=-10.941}
  [1678] = {j1=-10.945, j2=61.151, j3=49.616, j4=-3.905, j5=76.798, j6=-10.532}
  [1679] = {j1=-10.920, j2=61.658, j3=49.152, j4=-3.964, j5=77.158, j6=-10.101}
  [1680] = {j1=-10.896, j2=62.169, j3=48.681, j4=-4.023, j5=77.535, j6=-9.658}
  [1681] = {j1=-10.874, j2=62.679, j3=48.212, j4=-4.080, j5=77.918, j6=-9.211}
  [1682] = {j1=-10.854, j2=63.183, j3=47.753, j4=-4.132, j5=78.295, j6=-8.770}
  [1683] = {j1=-10.837, j2=63.675, j3=47.313, j4=-4.177, j5=78.655, j6=-8.342}
  [1684] = {j1=-10.823, j2=64.152, j3=46.900, j4=-4.214, j5=78.987, j6=-7.937}
  [1685] = {j1=-10.821, j2=64.233, j3=46.831, j4=-4.220, j5=79.041, j6=-7.869}
  [1686] = {j1=-10.804, j2=64.682, j3=46.465, j4=-4.272, j5=79.319, j6=-7.487}
  [1687] = {j1=-10.776, j2=65.166, j3=46.112, j4=-4.372, j5=79.552, j6=-7.071}
  [1688] = {j1=-10.740, j2=65.589, j3=45.875, j4=-4.513, j5=79.641, j6=-6.716}
  [1689] = {j1=-10.709, j2=65.879, j3=45.783, j4=-4.647, j5=79.583, j6=-6.493}
  [1690] = {j1=-10.678, j2=66.121, j3=45.778, j4=-4.786, j5=79.414, j6=-6.334}
  [1691] = {j1=-10.646, j2=66.321, j3=45.847, j4=-4.932, j5=79.147, j6=-6.232}
  [1692] = {j1=-10.614, j2=66.484, j3=45.981, j4=-5.090, j5=78.792, j6=-6.178}
  [1693] = {j1=-10.580, j2=66.614, j3=46.168, j4=-5.262, j5=78.363, j6=-6.165}
  [1694] = {j1=-10.543, j2=66.716, j3=46.397, j4=-5.453, j5=77.871, j6=-6.184}
  [1695] = {j1=-10.542, j2=66.735, j3=46.365, j4=-5.456, j5=77.930, j6=-6.141}
  [1696] = {j1=-10.579, j2=66.632, j3=46.137, j4=-5.265, j5=78.418, j6=-6.124}
  [1697] = {j1=-10.614, j2=66.500, j3=45.952, j4=-5.092, j5=78.844, j6=-6.139}
  [1698] = {j1=-10.646, j2=66.337, j3=45.820, j4=-4.933, j5=79.196, j6=-6.194}
  [1699] = {j1=-10.678, j2=66.136, j3=45.752, j4=-4.785, j5=79.461, j6=-6.297}
  [1700] = {j1=-10.709, j2=65.894, j3=45.758, j4=-4.646, j5=79.629, j6=-6.457}
  [1701] = {j1=-10.741, j2=65.603, j3=45.849, j4=-4.511, j5=79.686, j6=-6.681}
  [1702] = {j1=-10.777, j2=65.182, j3=46.086, j4=-4.368, j5=79.598, j6=-7.035}
  [1703] = {j1=-10.805, j2=64.697, j3=46.437, j4=-4.267, j5=79.366, j6=-7.450}
  [1704] = {j1=-10.822, j2=64.249, j3=46.803, j4=-4.215, j5=79.088, j6=-7.831}
  [1705] = {j1=-10.824, j2=64.168, j3=46.872, j4=-4.208, j5=79.034, j6=-7.900}
  [1706] = {j1=-10.838, j2=63.690, j3=47.287, j4=-4.172, j5=78.700, j6=-8.306}
  [1707] = {j1=-10.855, j2=63.197, j3=47.728, j4=-4.126, j5=78.337, j6=-8.735}
  [1708] = {j1=-10.876, j2=62.692, j3=48.189, j4=-4.074, j5=77.957, j6=-9.177}
  [1709] = {j1=-10.898, j2=62.180, j3=48.661, j4=-4.017, j5=77.571, j6=-9.625}
  [1710] = {j1=-10.922, j2=61.669, j3=49.133, j4=-3.958, j5=77.192, j6=-10.068}
  [1711] = {j1=-10.947, j2=61.162, j3=49.597, j4=-3.898, j5=76.832, j6=-10.499}
  [1712] = {j1=-10.972, j2=60.665, j3=50.042, j4=-3.840, j5=76.505, j6=-10.906}
  [1713] = {j1=-10.991, j2=60.244, j3=50.409, j4=-3.800, j5=76.253, j6=-11.233}
  [1714] = {j1=-11.005, j2=59.834, j3=50.755, j4=-3.777, j5=76.033, j6=-11.527}
  [1715] = {j1=-11.014, j2=59.435, j3=51.082, j4=-3.770, j5=75.839, j6=-11.794}
  [1716] = {j1=-11.019, j2=59.046, j3=51.392, j4=-3.777, j5=75.669, j6=-12.036}
  [1717] = {j1=-11.019, j2=59.031, j3=51.404, j4=-3.777, j5=75.662, j6=-12.044}
  [1718] = {j1=-11.020, j2=59.081, j3=51.315, j4=-3.772, j5=75.784, j6=-11.971}
  [1719] = {j1=-11.020, j2=59.095, j3=51.305, j4=-3.771, j5=75.789, j6=-11.963}
  [1720] = {j1=-11.015, j2=59.480, j3=51.003, j4=-3.764, j5=75.950, j6=-11.725}
  [1721] = {j1=-11.006, j2=59.873, j3=50.685, j4=-3.771, j5=76.133, j6=-11.464}
  [1722] = {j1=-10.992, j2=60.278, j3=50.348, j4=-3.793, j5=76.343, j6=-11.175}
  [1723] = {j1=-10.973, j2=60.695, j3=49.989, j4=-3.833, j5=76.585, j6=-10.853}
  [1724] = {j1=-10.949, j2=61.188, j3=49.550, j4=-3.891, j5=76.906, j6=-10.449}
  [1725] = {j1=-10.924, j2=61.694, j3=49.089, j4=-3.950, j5=77.263, j6=-10.019}
  [1726] = {j1=-10.900, j2=62.205, j3=48.618, j4=-4.009, j5=77.641, j6=-9.575}
  [1727] = {j1=-10.878, j2=62.716, j3=48.146, j4=-4.066, j5=78.028, j6=-9.126}
  [1728] = {j1=-10.857, j2=63.222, j3=47.684, j4=-4.118, j5=78.410, j6=-8.681}
  [1729] = {j1=-10.840, j2=63.716, j3=47.242, j4=-4.164, j5=78.773, j6=-8.251}
  [1730] = {j1=-10.826, j2=64.193, j3=46.829, j4=-4.201, j5=79.106, j6=-7.844}
  [1731] = {j1=-10.824, j2=64.273, j3=46.761, j4=-4.207, j5=79.159, j6=-7.776}
  [1732] = {j1=-10.807, j2=64.720, j3=46.398, j4=-4.260, j5=79.434, j6=-7.395}
  [1733] = {j1=-10.779, j2=65.202, j3=46.051, j4=-4.362, j5=79.661, j6=-6.981}
  [1734] = {j1=-10.742, j2=65.622, j3=45.818, j4=-4.506, j5=79.745, j6=-6.627}
  [1735] = {j1=-10.710, j2=65.911, j3=45.728, j4=-4.642, j5=79.686, j6=-6.403}
  [1736] = {j1=-10.678, j2=66.153, j3=45.724, j4=-4.784, j5=79.518, j6=-6.242}
  [1737] = {j1=-10.647, j2=66.353, j3=45.792, j4=-4.933, j5=79.253, j6=-6.136}
  [1738] = {j1=-10.614, j2=66.517, j3=45.924, j4=-5.092, j5=78.902, j6=-6.079}
  [1739] = {j1=-10.579, j2=66.648, j3=46.108, j4=-5.266, j5=78.478, j6=-6.061}
  [1740] = {j1=-10.542, j2=66.752, j3=46.335, j4=-5.459, j5=77.991, j6=-6.076}
  [1741] = {j1=-10.541, j2=66.780, j3=46.286, j4=-5.464, j5=78.080, j6=-6.011}
  [1742] = {j1=-10.578, j2=66.675, j3=46.061, j4=-5.270, j5=78.562, j6=-5.999}
  [1743] = {j1=-10.613, j2=66.543, j3=45.879, j4=-5.095, j5=78.983, j6=-6.019}
  [1744] = {j1=-10.646, j2=66.378, j3=45.749, j4=-4.934, j5=79.330, j6=-6.079}
  [1745] = {j1=-10.678, j2=66.177, j3=45.681, j4=-4.784, j5=79.592, j6=-6.186}
  [1746] = {j1=-10.710, j2=65.934, j3=45.687, j4=-4.641, j5=79.759, j6=-6.348}
  [1747] = {j1=-10.743, j2=65.645, j3=45.776, j4=-4.503, j5=79.817, j6=-6.573}
  [1748] = {j1=-10.780, j2=65.226, j3=46.008, j4=-4.357, j5=79.734, j6=-6.926}
  [1749] = {j1=-10.809, j2=64.746, j3=46.353, j4=-4.254, j5=79.509, j6=-7.340}
  [1750] = {j1=-10.826, j2=64.299, j3=46.715, j4=-4.200, j5=79.234, j6=-7.720}
  [1751] = {j1=-10.828, j2=64.218, j3=46.784, j4=-4.194, j5=79.180, j6=-7.788}
  [1752] = {j1=-10.842, j2=63.740, j3=47.199, j4=-4.156, j5=78.845, j6=-8.196}
  [1753] = {j1=-10.859, j2=63.245, j3=47.643, j4=-4.110, j5=78.478, j6=-8.628}
  [1754] = {j1=-10.880, j2=62.738, j3=48.107, j4=-4.057, j5=78.093, j6=-9.075}
  [1755] = {j1=-10.902, j2=62.226, j3=48.581, j4=-4.000, j5=77.703, j6=-9.525}
  [1756] = {j1=-10.926, j2=61.714, j3=49.054, j4=-3.941, j5=77.322, j6=-9.970}
  [1757] = {j1=-10.951, j2=61.208, j3=49.515, j4=-3.882, j5=76.966, j6=-10.398}
  [1758] = {j1=-10.975, j2=60.717, j3=49.950, j4=-3.824, j5=76.649, j6=-10.800}
  [1759] = {j1=-10.994, j2=60.303, j3=50.304, j4=-3.784, j5=76.412, j6=-11.118}
  [1760] = {j1=-11.008, j2=59.902, j3=50.635, j4=-3.762, j5=76.210, j6=-11.402}
  [1761] = {j1=-11.017, j2=59.512, j3=50.946, j4=-3.755, j5=76.034, j6=-11.657}
  [1762] = {j1=-11.021, j2=59.129, j3=51.243, j4=-3.763, j5=75.878, j6=-11.891}
  [1763] = {j1=-11.022, j2=59.115, j3=51.254, j4=-3.763, j5=75.872, j6=-11.899}
  [1764] = {j1=-11.022, j2=59.163, j3=51.170, j4=-3.758, j5=75.988, j6=-11.829}
  [1765] = {j1=-11.022, j2=59.176, j3=51.160, j4=-3.757, j5=75.992, j6=-11.821}
  [1766] = {j1=-11.018, j2=59.554, j3=50.870, j4=-3.749, j5=76.141, j6=-11.591}
  [1767] = {j1=-11.009, j2=59.940, j3=50.567, j4=-3.756, j5=76.307, j6=-11.340}
  [1768] = {j1=-10.996, j2=60.336, j3=50.245, j4=-3.778, j5=76.500, j6=-11.061}
  [1769] = {j1=-10.977, j2=60.747, j3=49.898, j4=-3.817, j5=76.729, j6=-10.747}
  [1770] = {j1=-10.953, j2=61.235, j3=49.468, j4=-3.874, j5=77.040, j6=-10.348}
  [1771] = {j1=-10.928, j2=61.739, j3=49.010, j4=-3.933, j5=77.393, j6=-9.920}
  [1772] = {j1=-10.904, j2=62.250, j3=48.539, j4=-3.992, j5=77.772, j6=-9.475}
  [1773] = {j1=-10.882, j2=62.763, j3=48.065, j4=-4.049, j5=78.162, j6=-9.023}
  [1774] = {j1=-10.861, j2=63.270, j3=47.600, j4=-4.102, j5=78.548, j6=-8.575}
  [1775] = {j1=-10.844, j2=63.765, j3=47.156, j4=-4.148, j5=78.915, j6=-8.142}
  [1776] = {j1=-10.830, j2=64.242, j3=46.743, j4=-4.186, j5=79.249, j6=-7.733}
  [1777] = {j1=-10.827, j2=64.322, j3=46.675, j4=-4.192, j5=79.302, j6=-7.665}
  [1778] = {j1=-10.810, j2=64.767, j3=46.316, j4=-4.246, j5=79.574, j6=-7.285}
  [1779] = {j1=-10.782, j2=65.246, j3=45.974, j4=-4.351, j5=79.796, j6=-6.872}
  [1780] = {j1=-10.744, j2=65.663, j3=45.745, j4=-4.498, j5=79.876, j6=-6.518}
  [1781] = {j1=-10.711, j2=65.951, j3=45.658, j4=-4.638, j5=79.815, j6=-6.292}
  [1782] = {j1=-10.679, j2=66.193, j3=45.654, j4=-4.782, j5=79.648, j6=-6.129}
  [1783] = {j1=-10.647, j2=66.394, j3=45.722, j4=-4.933, j5=79.386, j6=-6.020}
  [1784] = {j1=-10.613, j2=66.558, j3=45.852, j4=-5.095, j5=79.039, j6=-5.959}
  [1785] = {j1=-10.578, j2=66.691, j3=46.034, j4=-5.272, j5=78.620, j6=-5.937}
  [1786] = {j1=-10.540, j2=66.796, j3=46.259, j4=-5.466, j5=78.139, j6=-5.946}
  [1787] = {j1=-10.539, j2=66.824, j3=46.210, j4=-5.471, j5=78.227, j6=-5.882}
  [1788] = {j1=-10.577, j2=66.718, j3=45.987, j4=-5.275, j5=78.704, j6=-5.874}
  [1789] = {j1=-10.613, j2=66.585, j3=45.806, j4=-5.098, j5=79.120, j6=-5.898}
  [1790] = {j1=-10.647, j2=66.419, j3=45.678, j4=-4.935, j5=79.464, j6=-5.962}
  [1791] = {j1=-10.679, j2=66.218, j3=45.611, j4=-4.782, j5=79.724, j6=-6.072}
  [1792] = {j1=-10.712, j2=65.975, j3=45.616, j4=-4.636, j5=79.889, j6=-6.237}
  [1793] = {j1=-10.745, j2=65.687, j3=45.704, j4=-4.495, j5=79.948, j6=-6.463}
  [1794] = {j1=-10.783, j2=65.270, j3=45.931, j4=-4.346, j5=79.869, j6=-6.817}
  [1795] = {j1=-10.812, j2=64.792, j3=46.272, j4=-4.240, j5=79.647, j6=-7.230}
  [1796] = {j1=-10.829, j2=64.347, j3=46.632, j4=-4.185, j5=79.374, j6=-7.611}
  [1797] = {j1=-10.832, j2=64.266, j3=46.701, j4=-4.178, j5=79.320, j6=-7.679}
  [1798] = {j1=-10.846, j2=63.788, j3=47.115, j4=-4.140, j5=78.984, j6=-8.088}
  [1799] = {j1=-10.864, j2=63.292, j3=47.561, j4=-4.093, j5=78.614, j6=-8.523}
  [1800] = {j1=-10.884, j2=62.784, j3=48.028, j4=-4.040, j5=78.225, j6=-8.972}
  [1801] = {j1=-10.907, j2=62.270, j3=48.503, j4=-3.983, j5=77.833, j6=-9.425}
  [1802] = {j1=-10.931, j2=61.758, j3=48.976, j4=-3.924, j5=77.452, j6=-9.870}
  [1803] = {j1=-10.955, j2=61.255, j3=49.433, j4=-3.865, j5=77.099, j6=-10.297}
  [1804] = {j1=-10.979, j2=60.768, j3=49.861, j4=-3.808, j5=76.790, j6=-10.693}
  [1805] = {j1=-10.998, j2=60.359, j3=50.204, j4=-3.769, j5=76.566, j6=-11.004}
  [1806] = {j1=-11.011, j2=59.966, j3=50.521, j4=-3.747, j5=76.378, j6=-11.279}
  [1807] = {j1=-11.019, j2=59.583, j3=50.820, j4=-3.741, j5=76.217, j6=-11.526}
  [1808] = {j1=-11.024, j2=59.207, j3=51.106, j4=-3.749, j5=76.073, j6=-11.753}
  [1809] = {j1=-11.024, j2=59.193, j3=51.117, j4=-3.749, j5=76.068, j6=-11.761}
  [1810] = {j1=-11.024, j2=59.237, j3=51.038, j4=-3.744, j5=76.178, j6=-11.694}
  [1811] = {j1=-11.024, j2=59.250, j3=51.028, j4=-3.743, j5=76.182, j6=-11.686}
  [1812] = {j1=-11.020, j2=59.623, j3=50.748, j4=-3.735, j5=76.319, j6=-11.462}
  [1813] = {j1=-11.012, j2=60.002, j3=50.457, j4=-3.741, j5=76.472, j6=-11.218}
  [1814] = {j1=-10.999, j2=60.392, j3=50.146, j4=-3.762, j5=76.652, j6=-10.947}
  [1815] = {j1=-10.981, j2=60.797, j3=49.809, j4=-3.801, j5=76.869, j6=-10.640}
  [1816] = {j1=-10.957, j2=61.281, j3=49.386, j4=-3.858, j5=77.172, j6=-10.246}
  [1817] = {j1=-10.933, j2=61.783, j3=48.932, j4=-3.916, j5=77.522, j6=-9.820}
  [1818] = {j1=-10.909, j2=62.294, j3=48.461, j4=-3.975, j5=77.901, j6=-9.375}
  [1819] = {j1=-10.886, j2=62.807, j3=47.987, j4=-4.032, j5=78.293, j6=-8.921}
  [1820] = {j1=-10.866, j2=63.315, j3=47.521, j4=-4.085, j5=78.682, j6=-8.471}
  [1821] = {j1=-10.848, j2=63.811, j3=47.075, j4=-4.132, j5=79.051, j6=-8.035}
  [1822] = {j1=-10.834, j2=64.288, j3=46.662, j4=-4.171, j5=79.386, j6=-7.625}
  [1823] = {j1=-10.831, j2=64.368, j3=46.594, j4=-4.177, j5=79.439, j6=-7.556}
  [1824] = {j1=-10.814, j2=64.812, j3=46.237, j4=-4.233, j5=79.710, j6=-7.175}
  [1825] = {j1=-10.784, j2=65.289, j3=45.898, j4=-4.340, j5=79.929, j6=-6.762}
  [1826] = {j1=-10.746, j2=65.705, j3=45.673, j4=-4.490, j5=80.006, j6=-6.407}
  [1827] = {j1=-10.713, j2=65.992, j3=45.587, j4=-4.633, j5=79.945, j6=-6.180}
  [1828] = {j1=-10.680, j2=66.234, j3=45.584, j4=-4.779, j5=79.779, j6=-6.014}
  [1829] = {j1=-10.647, j2=66.435, j3=45.651, j4=-4.933, j5=79.519, j6=-5.903}
  [1830] = {j1=-10.613, j2=66.600, j3=45.781, j4=-5.098, j5=79.175, j6=-5.837}
  [1831] = {j1=-10.577, j2=66.733, j3=45.961, j4=-5.276, j5=78.760, j6=-5.811}
  [1832] = {j1=-10.539, j2=66.839, j3=46.184, j4=-5.473, j5=78.283, j6=-5.817}
  [1833] = {j1=-10.538, j2=66.868, j3=46.135, j4=-5.478, j5=78.371, j6=-5.752}
  [1834] = {j1=-10.577, j2=66.761, j3=45.914, j4=-5.280, j5=78.844, j6=-5.749}
  [1835] = {j1=-10.613, j2=66.626, j3=45.735, j4=-5.101, j5=79.257, j6=-5.777}
  [1836] = {j1=-10.647, j2=66.460, j3=45.607, j4=-4.935, j5=79.597, j6=-5.843}
  [1837] = {j1=-10.680, j2=66.259, j3=45.540, j4=-4.779, j5=79.856, j6=-5.956}
  [1838] = {j1=-10.713, j2=66.017, j3=45.544, j4=-4.631, j5=80.020, j6=-6.123}
  [1839] = {j1=-10.747, j2=65.729, j3=45.631, j4=-4.487, j5=80.079, j6=-6.352}
  [1840] = {j1=-10.786, j2=65.313, j3=45.856, j4=-4.334, j5=80.001, j6=-6.707}
  [1841] = {j1=-10.816, j2=64.836, j3=46.195, j4=-4.226, j5=79.781, j6=-7.121}
  [1842] = {j1=-10.833, j2=64.392, j3=46.553, j4=-4.170, j5=79.509, j6=-7.503}
  [1843] = {j1=-10.836, j2=64.311, j3=46.622, j4=-4.163, j5=79.454, j6=-7.571}
  [1844] = {j1=-10.850, j2=63.833, j3=47.037, j4=-4.124, j5=79.117, j6=-7.983}
  [1845] = {j1=-10.868, j2=63.336, j3=47.484, j4=-4.076, j5=78.745, j6=-8.419}
  [1846] = {j1=-10.889, j2=62.827, j3=47.951, j4=-4.023, j5=78.354, j6=-8.870}
  [1847] = {j1=-10.911, j2=62.313, j3=48.427, j4=-3.965, j5=77.960, j6=-9.324}
  [1848] = {j1=-10.935, j2=61.802, j3=48.899, j4=-3.907, j5=77.580, j6=-9.770}
  [1849] = {j1=-10.959, j2=61.301, j3=49.352, j4=-3.848, j5=77.230, j6=-10.194}
  [1850] = {j1=-10.983, j2=60.817, j3=49.774, j4=-3.792, j5=76.929, j6=-10.586}
  [1851] = {j1=-11.001, j2=60.414, j3=50.108, j4=-3.754, j5=76.714, j6=-10.891}
  [1852] = {j1=-11.014, j2=60.026, j3=50.415, j4=-3.732, j5=76.538, j6=-11.159}
  [1853] = {j1=-11.022, j2=59.649, j3=50.703, j4=-3.726, j5=76.388, j6=-11.400}
  [1854] = {j1=-11.026, j2=59.277, j3=50.981, j4=-3.734, j5=76.254, j6=-11.621}
  [1855] = {j1=-11.026, j2=59.263, j3=50.991, j4=-3.735, j5=76.248, j6=-11.629}
  [1856] = {j1=-11.027, j2=59.305, j3=50.917, j4=-3.730, j5=76.352, j6=-11.565}
  [1857] = {j1=-11.027, j2=59.318, j3=50.908, j4=-3.729, j5=76.356, j6=-11.558}
  [1858] = {j1=-11.023, j2=59.687, j3=50.636, j4=-3.721, j5=76.485, j6=-11.338}
  [1859] = {j1=-11.015, j2=60.061, j3=50.353, j4=-3.726, j5=76.628, j6=-11.100}
  [1860] = {j1=-11.003, j2=60.445, j3=50.052, j4=-3.747, j5=76.798, j6=-10.835}
  [1861] = {j1=-10.985, j2=60.846, j3=49.722, j4=-3.785, j5=77.007, j6=-10.533}
  [1862] = {j1=-10.961, j2=61.327, j3=49.305, j4=-3.841, j5=77.304, j6=-10.142}
  [1863] = {j1=-10.937, j2=61.827, j3=48.855, j4=-3.899, j5=77.650, j6=-9.719}
  [1864] = {j1=-10.913, j2=62.337, j3=48.386, j4=-3.957, j5=78.028, j6=-9.274}
  [1865] = {j1=-10.891, j2=62.850, j3=47.911, j4=-4.014, j5=78.420, j6=-8.820}
  [1866] = {j1=-10.870, j2=63.358, j3=47.445, j4=-4.068, j5=78.810, j6=-8.368}
  [1867] = {j1=-10.852, j2=63.854, j3=46.999, j4=-4.116, j5=79.181, j6=-7.930}
  [1868] = {j1=-10.838, j2=64.331, j3=46.586, j4=-4.155, j5=79.517, j6=-7.518}
  [1869] = {j1=-10.835, j2=64.412, j3=46.518, j4=-4.161, j5=79.570, j6=-7.449}
  [1870] = {j1=-10.818, j2=64.855, j3=46.162, j4=-4.218, j5=79.841, j6=-7.067}
  [1871] = {j1=-10.787, j2=65.332, j3=45.824, j4=-4.328, j5=80.059, j6=-6.652}
  [1872] = {j1=-10.749, j2=65.746, j3=45.601, j4=-4.482, j5=80.136, j6=-6.295}
  [1873] = {j1=-10.714, j2=66.033, j3=45.516, j4=-4.627, j5=80.075, j6=-6.066}
  [1874] = {j1=-10.681, j2=66.274, j3=45.513, j4=-4.777, j5=79.910, j6=-5.898}
  [1875] = {j1=-10.647, j2=66.475, j3=45.581, j4=-4.933, j5=79.651, j6=-5.783}
  [1876] = {j1=-10.613, j2=66.641, j3=45.710, j4=-5.100, j5=79.310, j6=-5.715}
  [1877] = {j1=-10.577, j2=66.775, j3=45.890, j4=-5.281, j5=78.897, j6=-5.686}
  [1878] = {j1=-10.538, j2=66.881, j3=46.112, j4=-5.479, j5=78.425, j6=-5.687}
  [1879] = {j1=-10.537, j2=66.910, j3=46.063, j4=-5.484, j5=78.513, j6=-5.623}
  [1880] = {j1=-10.576, j2=66.802, j3=45.842, j4=-5.285, j5=78.982, j6=-5.623}
  [1881] = {j1=-10.612, j2=66.667, j3=45.664, j4=-5.103, j5=79.392, j6=-5.654}
  [1882] = {j1=-10.647, j2=66.501, j3=45.536, j4=-4.935, j5=79.731, j6=-5.723}
  [1883] = {j1=-10.681, j2=66.300, j3=45.469, j4=-4.777, j5=79.988, j6=-5.839}
  [1884] = {j1=-10.715, j2=66.058, j3=45.473, j4=-4.626, j5=80.151, j6=-6.008}
  [1885] = {j1=-10.749, j2=65.771, j3=45.558, j4=-4.479, j5=80.210, j6=-6.239}
  [1886] = {j1=-10.789, j2=65.355, j3=45.783, j4=-4.323, j5=80.131, j6=-6.597}
  [1887] = {j1=-10.819, j2=64.878, j3=46.121, j4=-4.212, j5=79.910, j6=-7.013}
  [1888] = {j1=-10.837, j2=64.434, j3=46.479, j4=-4.154, j5=79.637, j6=-7.397}
  [1889] = {j1=-10.840, j2=64.353, j3=46.548, j4=-4.147, j5=79.582, j6=-7.465}
  [1890] = {j1=-10.854, j2=63.875, j3=46.963, j4=-4.107, j5=79.244, j6=-7.878}
  [1891] = {j1=-10.873, j2=63.378, j3=47.410, j4=-4.059, j5=78.871, j6=-8.317}
  [1892] = {j1=-10.893, j2=62.869, j3=47.878, j4=-4.005, j5=78.479, j6=-8.769}
  [1893] = {j1=-10.916, j2=62.356, j3=48.353, j4=-3.948, j5=78.085, j6=-9.223}
  [1894] = {j1=-10.940, j2=61.845, j3=48.822, j4=-3.889, j5=77.706, j6=-9.668}
  [1895] = {j1=-10.964, j2=61.346, j3=49.272, j4=-3.831, j5=77.360, j6=-10.090}
  [1896] = {j1=-10.987, j2=60.865, j3=49.689, j4=-3.776, j5=77.064, j6=-10.479}
  [1897] = {j1=-11.005, j2=60.465, j3=50.017, j4=-3.738, j5=76.857, j6=-10.779}
  [1898] = {j1=-11.017, j2=60.082, j3=50.316, j4=-3.717, j5=76.689, j6=-11.042}
  [1899] = {j1=-11.025, j2=59.709, j3=50.597, j4=-3.712, j5=76.547, j6=-11.278}
  [1900] = {j1=-11.029, j2=59.341, j3=50.868, j4=-3.720, j5=76.420, j6=-11.496}
  [1901] = {j1=-11.029, j2=59.327, j3=50.878, j4=-3.720, j5=76.414, j6=-11.504}
  [1902] = {j1=-11.030, j2=59.366, j3=50.809, j4=-3.715, j5=76.512, j6=-11.443}
  [1903] = {j1=-11.030, j2=59.379, j3=50.800, j4=-3.715, j5=76.516, j6=-11.436}
  [1904] = {j1=-11.026, j2=59.745, j3=50.533, j4=-3.706, j5=76.639, j6=-11.220}
  [1905] = {j1=-11.018, j2=60.115, j3=50.257, j4=-3.712, j5=76.775, j6=-10.985}
  [1906] = {j1=-11.006, j2=60.496, j3=49.962, j4=-3.732, j5=76.939, j6=-10.724}
  [1907] = {j1=-10.989, j2=60.894, j3=49.638, j4=-3.769, j5=77.142, j6=-10.425}
  [1908] = {j1=-10.965, j2=61.372, j3=49.225, j4=-3.824, j5=77.434, j6=-10.038}
  [1909] = {j1=-10.942, j2=61.870, j3=48.779, j4=-3.881, j5=77.776, j6=-9.617}
  [1910] = {j1=-10.918, j2=62.379, j3=48.312, j4=-3.939, j5=78.152, j6=-9.173}
  [1911] = {j1=-10.895, j2=62.891, j3=47.839, j4=-3.997, j5=78.543, j6=-8.718}
  [1912] = {j1=-10.875, j2=63.399, j3=47.374, j4=-4.050, j5=78.933, j6=-8.266}
  [1913] = {j1=-10.857, j2=63.895, j3=46.928, j4=-4.099, j5=79.305, j6=-7.827}
  [1914] = {j1=-10.842, j2=64.372, j3=46.515, j4=-4.139, j5=79.642, j6=-7.413}
  [1915] = {j1=-10.839, j2=64.452, j3=46.447, j4=-4.146, j5=79.695, j6=-7.344}
  [1916] = {j1=-10.821, j2=64.896, j3=46.090, j4=-4.204, j5=79.967, j6=-6.960}
  [1917] = {j1=-10.791, j2=65.373, j3=45.753, j4=-4.316, j5=80.187, j6=-6.542}
  [1918] = {j1=-10.751, j2=65.788, j3=45.530, j4=-4.474, j5=80.266, j6=-6.182}
  [1919] = {j1=-10.716, j2=66.074, j3=45.445, j4=-4.622, j5=80.206, j6=-5.950}
  [1920] = {j1=-10.682, j2=66.315, j3=45.443, j4=-4.774, j5=80.041, j6=-5.779}
  [1921] = {j1=-10.648, j2=66.516, j3=45.511, j4=-4.933, j5=79.783, j6=-5.662}
  [1922] = {j1=-10.613, j2=66.681, j3=45.640, j4=-5.102, j5=79.443, j6=-5.592}
  [1923] = {j1=-10.576, j2=66.815, j3=45.820, j4=-5.285, j5=79.033, j6=-5.560}
  [1924] = {j1=-10.537, j2=66.922, j3=46.041, j4=-5.485, j5=78.563, j6=-5.558}
  [1925] = {j1=-10.536, j2=66.950, j3=45.992, j4=-5.490, j5=78.652, j6=-5.493}
  [1926] = {j1=-10.575, j2=66.842, j3=45.772, j4=-5.288, j5=79.118, j6=-5.497}
  [1927] = {j1=-10.612, j2=66.708, j3=45.593, j4=-5.104, j5=79.526, j6=-5.530}
  [1928] = {j1=-10.647, j2=66.542, j3=45.465, j4=-4.934, j5=79.864, j6=-5.601}
  [1929] = {j1=-10.682, j2=66.341, j3=45.397, j4=-4.774, j5=80.120, j6=-5.719}
  [1930] = {j1=-10.716, j2=66.099, j3=45.401, j4=-4.620, j5=80.282, j6=-5.891}
  [1931] = {j1=-10.752, j2=65.812, j3=45.487, j4=-4.470, j5=80.339, j6=-6.124}
  [1932] = {j1=-10.792, j2=65.396, j3=45.712, j4=-4.311, j5=80.258, j6=-6.486}
  [1933] = {j1=-10.823, j2=64.918, j3=46.051, j4=-4.197, j5=80.034, j6=-6.906}
  [1934] = {j1=-10.841, j2=64.474, j3=46.411, j4=-4.138, j5=79.759, j6=-7.292}
  [1935] = {j1=-10.844, j2=64.392, j3=46.479, j4=-4.131, j5=79.704, j6=-7.361}
  [1936] = {j1=-10.859, j2=63.914, j3=46.895, j4=-4.090, j5=79.364, j6=-7.776}
  [1937] = {j1=-10.877, j2=63.417, j3=47.342, j4=-4.041, j5=78.991, j6=-8.216}
  [1938] = {j1=-10.898, j2=62.909, j3=47.808, j4=-3.987, j5=78.600, j6=-8.668}
  [1939] = {j1=-10.921, j2=62.397, j3=48.281, j4=-3.930, j5=78.207, j6=-9.122}
  [1940] = {j1=-10.944, j2=61.888, j3=48.748, j4=-3.871, j5=77.831, j6=-9.565}
  [1941] = {j1=-10.968, j2=61.390, j3=49.194, j4=-3.814, j5=77.488, j6=-9.985}
  [1942] = {j1=-10.991, j2=60.912, j3=49.606, j4=-3.760, j5=77.197, j6=-10.371}
  [1943] = {j1=-11.008, j2=60.515, j3=49.930, j4=-3.723, j5=76.994, j6=-10.669}
  [1944] = {j1=-11.021, j2=60.133, j3=50.225, j4=-3.702, j5=76.830, j6=-10.929}
  [1945] = {j1=-11.028, j2=59.763, j3=50.501, j4=-3.697, j5=76.694, j6=-11.162}
  [1946] = {j1=-11.032, j2=59.398, j3=50.767, j4=-3.706, j5=76.570, j6=-11.378}
  [1947] = {j1=-11.032, j2=59.384, j3=50.778, j4=-3.706, j5=76.565, j6=-11.385}
  [1948] = {j1=-11.033, j2=59.421, j3=50.713, j4=-3.701, j5=76.657, j6=-11.328}
  [1949] = {j1=-11.033, j2=59.433, j3=50.705, j4=-3.700, j5=76.661, j6=-11.321}
  [1950] = {j1=-11.029, j2=59.797, j3=50.441, j4=-3.692, j5=76.780, j6=-11.106}
  [1951] = {j1=-11.022, j2=60.165, j3=50.169, j4=-3.697, j5=76.914, j6=-10.874}
  [1952] = {j1=-11.010, j2=60.545, j3=49.876, j4=-3.716, j5=77.074, j6=-10.614}
  [1953] = {j1=-10.993, j2=60.941, j3=49.556, j4=-3.753, j5=77.274, j6=-10.317}
  [1954] = {j1=-10.970, j2=61.417, j3=49.147, j4=-3.807, j5=77.562, j6=-9.932}
  [1955] = {j1=-10.946, j2=61.913, j3=48.704, j4=-3.863, j5=77.901, j6=-9.513}
  [1956] = {j1=-10.923, j2=62.419, j3=48.241, j4=-3.921, j5=78.274, j6=-9.071}
  [1957] = {j1=-10.900, j2=62.930, j3=47.771, j4=-3.978, j5=78.662, j6=-8.618}
  [1958] = {j1=-10.879, j2=63.437, j3=47.307, j4=-4.033, j5=79.051, j6=-8.165}
  [1959] = {j1=-10.861, j2=63.932, j3=46.863, j4=-4.081, j5=79.422, j6=-7.726}
  [1960] = {j1=-10.846, j2=64.410, j3=46.449, j4=-4.122, j5=79.760, j6=-7.310}
  [1961] = {j1=-10.844, j2=64.490, j3=46.381, j4=-4.129, j5=79.814, j6=-7.241}
  [1962] = {j1=-10.825, j2=64.935, j3=46.023, j4=-4.189, j5=80.089, j6=-6.853}
  [1963] = {j1=-10.794, j2=65.413, j3=45.683, j4=-4.304, j5=80.313, j6=-6.431}
  [1964] = {j1=-10.753, j2=65.828, j3=45.459, j4=-4.465, j5=80.394, j6=-6.066}
  [1965] = {j1=-10.717, j2=66.115, j3=45.374, j4=-4.616, j5=80.336, j6=-5.831}
  [1966] = {j1=-10.682, j2=66.356, j3=45.372, j4=-4.771, j5=80.172, j6=-5.659}
  [1967] = {j1=-10.648, j2=66.556, j3=45.442, j4=-4.932, j5=79.915, j6=-5.540}
  [1968] = {j1=-10.612, j2=66.721, j3=45.572, j4=-5.103, j5=79.575, j6=-5.467}
  [1969] = {j1=-10.575, j2=66.854, j3=45.752, j4=-5.288, j5=79.166, j6=-5.433}
  [1970] = {j1=-10.536, j2=66.962, j3=45.973, j4=-5.491, j5=78.699, j6=-5.428}
  [1971] = {j1=-10.535, j2=66.990, j3=45.924, j4=-5.496, j5=78.787, j6=-5.364}
  [1972] = {j1=-10.575, j2=66.882, j3=45.704, j4=-5.292, j5=79.252, j6=-5.370}
  [1973] = {j1=-10.612, j2=66.748, j3=45.524, j4=-5.106, j5=79.659, j6=-5.405}
  [1974] = {j1=-10.648, j2=66.583, j3=45.395, j4=-4.933, j5=79.996, j6=-5.478}
  [1975] = {j1=-10.683, j2=66.382, j3=45.326, j4=-4.770, j5=80.252, j6=-5.598}
  [1976] = {j1=-10.718, j2=66.141, j3=45.329, j4=-4.614, j5=80.413, j6=-5.772}
  [1977] = {j1=-10.754, j2=65.853, j3=45.415, j4=-4.461, j5=80.468, j6=-6.008}
  [1978] = {j1=-10.795, j2=65.436, j3=45.643, j4=-4.298, j5=80.382, j6=-6.375}
  [1979] = {j1=-10.827, j2=64.956, j3=45.985, j4=-4.182, j5=80.154, j6=-6.800}
  [1980] = {j1=-10.846, j2=64.510, j3=46.347, j4=-4.121, j5=79.875, j6=-7.190}
  [1981] = {j1=-10.848, j2=64.429, j3=46.416, j4=-4.114, j5=79.819, j6=-7.259}
  [1982] = {j1=-10.864, j2=63.950, j3=46.832, j4=-4.072, j5=79.478, j6=-7.676}
  [1983] = {j1=-10.882, j2=63.454, j3=47.277, j4=-4.023, j5=79.105, j6=-8.116}
  [1984] = {j1=-10.903, j2=62.947, j3=47.741, j4=-3.969, j5=78.716, j6=-8.567}
  [1985] = {j1=-10.925, j2=62.436, j3=48.211, j4=-3.912, j5=78.327, j6=-9.020}
  [1986] = {j1=-10.949, j2=61.930, j3=48.674, j4=-3.854, j5=77.954, j6=-9.461}
  [1987] = {j1=-10.972, j2=61.434, j3=49.117, j4=-3.797, j5=77.615, j6=-9.879}
  [1988] = {j1=-10.995, j2=60.958, j3=49.526, j4=-3.743, j5=77.326, j6=-10.263}
  [1989] = {j1=-11.012, j2=60.561, j3=49.848, j4=-3.707, j5=77.125, j6=-10.559}
  [1990] = {j1=-11.024, j2=60.181, j3=50.141, j4=-3.687, j5=76.963, j6=-10.819}
  [1991] = {j1=-11.032, j2=59.811, j3=50.415, j4=-3.682, j5=76.827, j6=-11.052}
  [1992] = {j1=-11.036, j2=59.448, j3=50.680, j4=-3.691, j5=76.706, j6=-11.266}
  [1993] = {j1=-11.036, j2=59.434, j3=50.690, j4=-3.691, j5=76.701, j6=-11.274}
  [1994] = {j1=-11.036, j2=59.468, j3=50.631, j4=-3.686, j5=76.787, j6=-11.220}
  [1995] = {j1=-11.036, j2=59.480, j3=50.622, j4=-3.686, j5=76.790, j6=-11.213}
  [1996] = {j1=-11.033, j2=59.843, j3=50.360, j4=-3.677, j5=76.909, j6=-10.998}
  [1997] = {j1=-11.026, j2=60.211, j3=50.088, j4=-3.681, j5=77.043, j6=-10.765}
  [1998] = {j1=-11.014, j2=60.591, j3=49.796, j4=-3.701, j5=77.203, j6=-10.505}
  [1999] = {j1=-10.997, j2=60.986, j3=49.476, j4=-3.736, j5=77.403, j6=-10.209}
  [2000] = {j1=-10.974, j2=61.461, j3=49.070, j4=-3.789, j5=77.689, j6=-9.826}
public mdesc mNomSpeed = {accel=100, vel=100, decel=100, tmax=99999, rmax=99999, blend=off, leave=50, reach=50}
public mdesc mdJointBlend = {accel=250, vel=30, decel=150, tmax=99999, rmax=99999, blend=off, leave=0, reach=0}
public mdesc mdLineBlend = {accel=80, vel=30, decel=30, tmax=763.92, rmax=9999, blend=joint, leave=0.1, reach=0.1}
public tool tTool = {x=968.000, y=-155.000, z=-238.000, rx=-90.000, ry=0.000, rz=180.000, fatherId=flange[0], ioLink=valve1}
